// TIA Portal V17 export
// export: Created 2023-04-11T09:33:39.3970323Z, ExportSetting WithDefaults, DisplayName Totally Integrated Automation Portal, DisplayVersion V17 Update 3, DisplayName TIA Portal Openness, DisplayVersion V17 Update 3, DisplayName TIA Portal Version Control Interface, DisplayVersion V17, DisplayName SINAMICS Startdrive Advanced, DisplayVersion V17 Update2, DisplayName SINAMICS Startdrive G130, G150, S120, S150, SINAMICS MV, S210, DisplayVersion V17 Update2, DisplayName SINAMICS Startdrive G110M, G120, G120C, G120D, G120P, G115D, DisplayVersion V17 Update2, DisplayName STEP 7 Professional, DisplayVersion V17 Update 3, DisplayName STEP 7 Safety, DisplayVersion V17, DisplayName WinCC UA Professional, DisplayVersion V17 Update 3
FUNCTION_BLOCK "FB_Pos_Check"   // FB55, LAD
{ S7_Optimized_Access := 'TRUE' }
VERSION : 0.1
// stored: AutoNumber true, IsIECCheckEnabled false, IsRetainMemResEnabled false, MemoryReserve 100, SetENOAutomatically false, UDAEnableTagReadback false
   VAR_INPUT
      Actual_Pos : DInt;
      Desired_Pos : DInt;
   END_VAR
   VAR_OUTPUT
      InPosition : Bool;
   END_VAR
   VAR
      Position_Dly { S7_SetPoint := 'True'} : TON_TIME;
   END_VAR
   VAR_TEMP
      Min : DInt;
      Max : DInt;
   END_VAR
BEGIN

REGION Network 1: Detect position
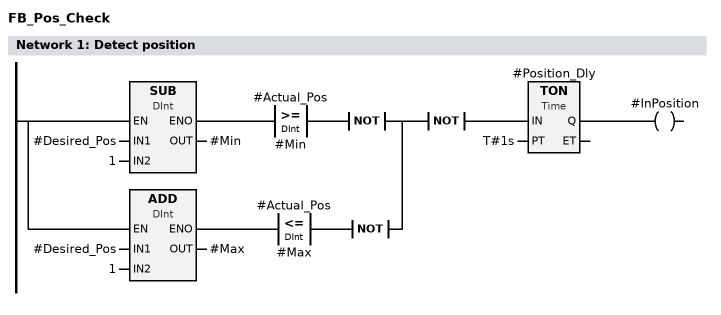
   RUNG wire#powerrail
      { S7_Templates := "SrcType := DInt" } Sub(in1 := #Desired_Pos, in2 := 1, out => #Min)
      { S7_Templates := "SrcType := DInt" } GE_Contact(in1 := #Actual_Pos, in2 := #Min)
      Not()
      wire#w1
      Not()
      { S7_Templates := "time_type := Time" } #Position_Dly.TON(pt := T#1s, et =>)
      Coil( #InPosition )
   END_RUNG
   RUNG wire#powerrail
      { S7_Templates := "SrcType := DInt" } Add(in1 := #Desired_Pos, in2 := 1, out => #Max)
      { S7_Templates := "SrcType := DInt" } LE_Contact(in1 := #Actual_Pos, in2 := #Max)
      Not()
   END_RUNG wire#w1
   // the same network as SCL:
   #Min := #Desired_Pos - 1;
   #Max := #Desired_Pos + 1;
   #Position_Dly(IN := NOT (NOT (#Actual_Pos >= #Min) OR NOT (#Actual_Pos <= #Max)), PT := T#1s);   // TON
   #InPosition := #Position_Dly.Q;
END_REGION
END_FUNCTION_BLOCK
